INTERFACE I_Action EXTENDS I_Object

METHOD Execute
VAR_INPUT
    ipObject: I_Object;
END_VAR
END_METHOD

END_INTERFACE

(* stored: Version 1.1.0.1, ProductVersion 3.1.4024.12
   Itf I_Action: Id {693c0bbf-2f16-0239-1f37-9574a10a96e2}
   Method Execute: Id {75b9d855-fb9c-05fc-252d-ef3f7519ed88} *)
